FUNCTION_BLOCK FB_InitializeControl
VAR
	_passed: BOOL;
	_initList: ARRAY [1..INITIALIZE.MAX_INIT_LIST] OF BOOL;
	_headerText: STRING;
	_totalCounter: INT;
	_passedCounter: INT;
	_failedCounter: INT;
END_VAR

METHOD Footer
ADSLOGSTR(msgCtrlMask := ADSLOG_MSGTYPE_ERROR, msgFmtStr := 'Total Tests: %s', TO_STRING(_totalCounter));
ADSLOGSTR(msgCtrlMask := ADSLOG_MSGTYPE_ERROR, msgFmtStr := 'Passed: %s', TO_STRING(_passedCounter));
ADSLOGSTR(msgCtrlMask := ADSLOG_MSGTYPE_ERROR, msgFmtStr := 'Failed: %s', TO_STRING(_failedCounter));
END_METHOD

METHOD Header
VAR_INPUT
	title: STRING;
END_VAR
_headerText := CONCAT('==========', title);
_headerText := CONCAT(_headerText, ' INITIALIZING==========');

ADSLOGSTR(ADSLOG_MSGTYPE_ERROR, _headerText, '');
END_METHOD

PROPERTY Passed : BOOL
GET
Passed := _passed;
END_GET
SET
IF _totalCounter >= MAX_INIT_LIST THEN
	RETURN;
END_IF

_totalCounter := _totalCounter + 1;

IF Passed THEN
	_passedCounter := _passedCounter + 1;
ELSE
	_failedCounter := _failedCounter + 1;
END_IF

_initList[_totalCounter] := Passed;

_passed := Passed AND _passed;
END_SET
END_PROPERTY

END_FUNCTION_BLOCK

(* stored: Version 1.1.0.1, ProductVersion 3.1.4024.10
   POU FB_InitializeControl: Id {421fb946-2c15-47dd-b9c5-885068f850a4}, SpecialFunc None
   Method Footer: Id {08800716-2bb4-4597-bfa2-2205d1cbf566}
   Method Header: Id {9088245b-b307-400b-a9a2-88e630daa675}
   Property Passed: Id {4491a244-136b-45b5-a40e-f803860d998b}
   Get Get: Id {9eb3beb3-2df0-4637-96aa-fce1eb278635}
   Set Set: Id {a5f5a565-0654-4c7f-b83a-fac76106764e} *)
